FUNCTION_BLOCK VFD_WRITE
VAR
  	fbWriteRegs : FB_MBWriteRegs; //Function call
	ipAddr      : STRING(15) := '192.168.1.5'; //IPADDRESS
  	M0 AT%MB0   : ARRAY [0..1] OF WORD;
  	startValue  : ARRAY [0..1] OF WORD;
	stopValue	: ARRAY [0..1] OF WORD;
	eWriteState	: (WAIT, START, STOP, WRITE); //state machine
	startTrigger 	: R_TRIG; //Trigger function block
	stopTrigger 	: R_TRIG; //Trigger function block
	Light AT %Q*: BOOL;
END_VAR

startValue[0] := INT_TO_WORD(18);
startValue[1] := INT_TO_WORD(4000);
stopValue[0] := INT_TO_WORD(1);
stopValue[1] := INT_TO_WORD(0);

startTrigger();
stopTrigger();
IF startTrigger.Q THEN
	IF eWriteState = WAIT THEN
		eWriteState := START;
	END_IF
END_IF

IF stopTrigger.Q THEN
	IF eWriteState = WAIT THEN
		eWriteState := STOP;
	END_IF
END_IF

CASE eWriteState OF
	WAIT: 
		//Do nothing
		
	START:
		fbWriteRegs(
			sIPAddr:= ipAddr, 
			nTCPPort:= 502, 
			nUnitID:= 16#FF, 
			nQuantity:= 2, 
			nMBAddr:= 16#2000, 
			cbLength:= SIZEOF(startValue), 
			pSrcAddr:= ADR(startValue), 
			bExecute:= TRUE, 
			tTimeout:= , 
			bBusy=> , 
			bError=> , 
			nErrId=> );
		
		eWriteState := WRITE;
		
	STOP:
		fbWriteRegs(
			sIPAddr:= ipAddr, 
			nTCPPort:= 502, 
			nUnitID:= 16#FF, 
			nQuantity:= 2, 
			nMBAddr:= 16#2000, 
			cbLength:= SIZEOF(stopValue), 
			pSrcAddr:= ADR(stopValue), 
			bExecute:= TRUE, 
			tTimeout:= , 
			bBusy=> , 
			bError=> , 
			nErrId=> );
		
		eWriteState := WRITE;
		
	WRITE :
		fbWriteRegs(bExecute := FALSE);
		IF NOT fbWriteRegs.bBusy OR fbWriteRegs.bError THEN
			eWriteState := WAIT;
		END_IF
		
		// 
END_CASE

END_FUNCTION_BLOCK

(* stored: Version 1.1.0.1, ProductVersion 3.1.4024.12
   POU VFD_WRITE: Id {8cbf1fd6-2d39-40a7-8131-7eca32614bdb}, SpecialFunc None *)
